// TIA Portal V15.1 export
// export: Created 2020-06-12T07:35:49.8818359Z, ExportSetting None, DisplayName Totally Integrated Automation Portal, DisplayVersion V15.1, DisplayName TIA Portal Openness, DisplayVersion V15.1, DisplayName STEP 7 Professional, DisplayVersion V15.1, DisplayName STEP 7 Safety, DisplayVersion V15.1, DisplayName WinCC Advanced, DisplayVersion V15.1
FUNCTION_BLOCK "MELT_PHASES_S"   // FB221, GRAPH
TITLE = S7GRAPH V5.0 FB
{ S7_Optimized_Access := 'TRUE' }
// Block comment
// stored: AcknowledgeErrorsRequired false, GraphVersion 2.0, LanguageInNetworks FBD, SetENOAutomatically false, WithAlarmHandling false
   // inherited from GRAPH_BASE
   VAR_INPUT
      INIT_SQ : Bool;
      eStart { ExternalAccessible := 'False'; ExternalVisible := 'False'; ExternalWritable := 'False'} : Bool;
      eCancel { ExternalAccessible := 'False'; ExternalVisible := 'False'; ExternalWritable := 'False'} : Bool;
      ePrepared { ExternalAccessible := 'False'; ExternalVisible := 'False'; ExternalWritable := 'False'} : Bool;
      ePause { ExternalAccessible := 'False'; ExternalVisible := 'False'; ExternalWritable := 'False'} : Bool;
      eStop { ExternalAccessible := 'False'; ExternalVisible := 'False'; ExternalWritable := 'False'} : Bool;
      eStarted { ExternalAccessible := 'False'; ExternalVisible := 'False'; ExternalWritable := 'False'} : Bool;
      eForceMT { ExternalAccessible := 'False'; ExternalVisible := 'False'; ExternalWritable := 'False'} : Bool;
      eStartHT { ExternalAccessible := 'False'; ExternalVisible := 'False'; ExternalWritable := 'False'} : Bool;
      eSlagMolten { ExternalAccessible := 'False'; ExternalVisible := 'False'; ExternalWritable := 'False'} : Bool;
      iCurrentRuns { ExternalAccessible := 'False'; ExternalVisible := 'False'; ExternalWritable := 'False'} : Bool;
      pStartDuration { ExternalAccessible := 'False'; ExternalVisible := 'False'; ExternalWritable := 'False'} : Int := 30;
      pHTDuration { ExternalAccessible := 'False'; ExternalVisible := 'False'; ExternalWritable := 'False'} : Int := 30;
   END_VAR
   VAR_OUTPUT
      qSTPhaseTime { ExternalAccessible := 'False'; ExternalVisible := 'False'; ExternalWritable := 'False'} : Real;   // stat phase actual time
      qHTPhaseTime { ExternalAccessible := 'False'; ExternalVisible := 'False'; ExternalWritable := 'False'} : Real;   // hottoping phase actual time
      qPhaseId { ExternalAccessible := 'False'; ExternalVisible := 'False'; ExternalWritable := 'False'} : Int;   // phase ID
   END_VAR
   VAR_IN_OUT
      ioPremelt { ExternalAccessible := 'False'; ExternalVisible := 'False'; ExternalWritable := 'False'} : Bool;
      ioMelting { ExternalAccessible := 'False'; ExternalVisible := 'False'; ExternalWritable := 'False'} : Bool;
      ioStartPhaseRun { ExternalAccessible := 'False'; ExternalVisible := 'False'; ExternalWritable := 'False'} : Bool;
      ioMainPhaseRun { ExternalAccessible := 'False'; ExternalVisible := 'False'; ExternalWritable := 'False'} : Bool;
      ioHTPhaseRun { ExternalAccessible := 'False'; ExternalVisible := 'False'; ExternalWritable := 'False'} : Bool;
      ioEnd { ExternalAccessible := 'False'; ExternalVisible := 'False'; ExternalWritable := 'False'} : Bool;
      ioStartPhaseDone { ExternalAccessible := 'False'; ExternalVisible := 'False'; ExternalWritable := 'False'} : Bool;
      ioMainPhaseDone { ExternalAccessible := 'False'; ExternalVisible := 'False'; ExternalWritable := 'False'} : Bool;
      ioHTPhaseDone { ExternalAccessible := 'False'; ExternalVisible := 'False'; ExternalWritable := 'False'} : Bool;
      ioPause { ExternalAccessible := 'False'; ExternalVisible := 'False'; ExternalWritable := 'False'} : Bool;
   END_VAR
   VAR
      sSlagMolten : Bool;
      sPhaseId { ExternalAccessible := 'False'; ExternalVisible := 'False'; ExternalWritable := 'False'} : SInt;
   END_VAR
   VAR_TEMP
      tStartPhaseDuration : Time;
      tHTPhaseDuration : Time;
      tVarR1 : Real;
      tPauseOn : Bool;
      tPauseOff : Bool;
      tSTPauseLockTime : DInt;
   END_VAR
BEGIN
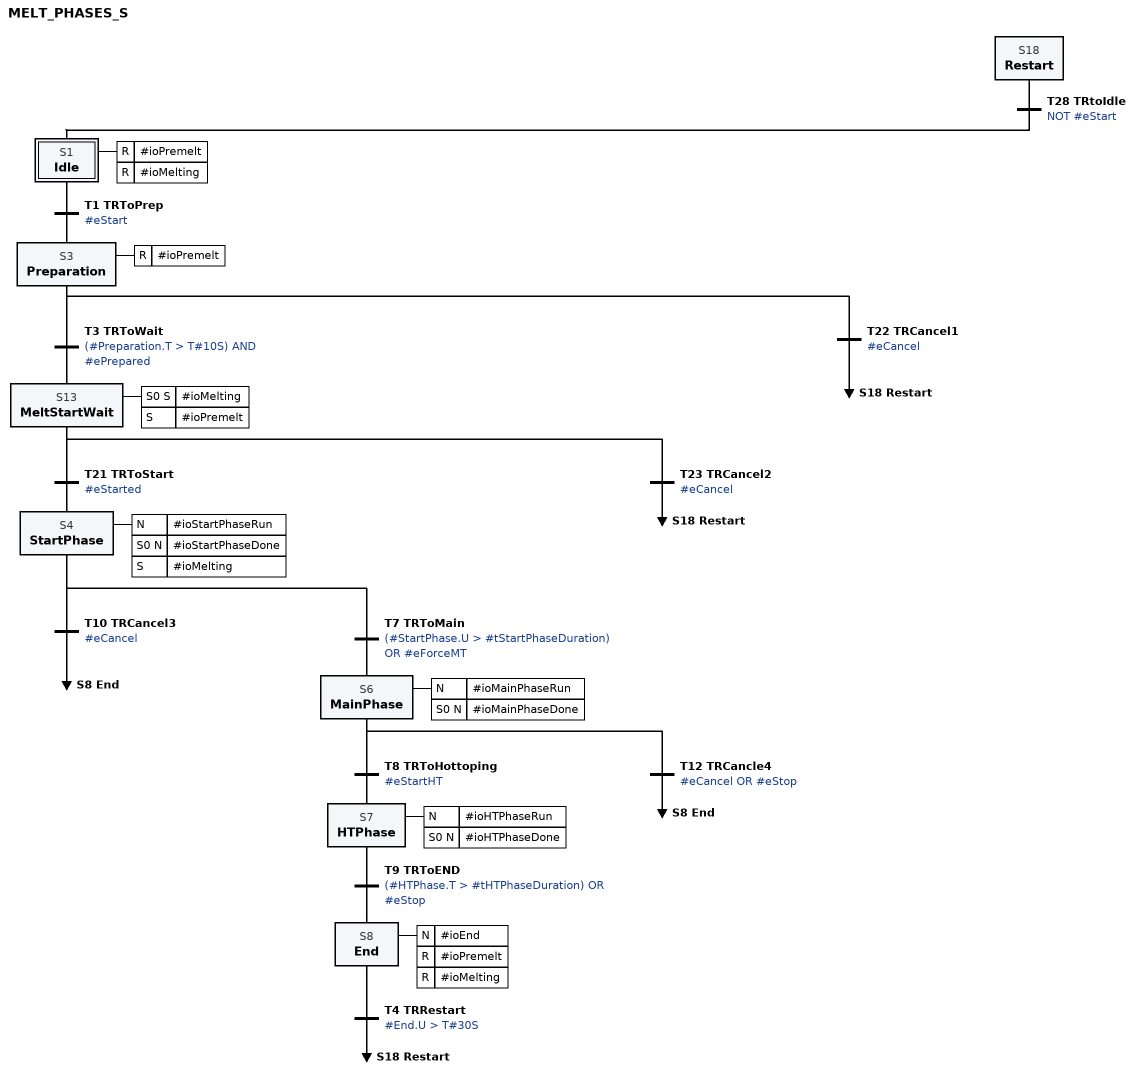
   // permanent pre-instructions
   NETWORK 1
   TITLE = Convert durations
      #tStartPhaseDuration := #pStartDuration * 60000;
      #tSTPauseLockTime := #tStartPhaseDuration / 10;
      #tHTPhaseDuration := #pHTDuration * 60000;
   NETWORK 2
   TITLE = Pause
      #tPauseOn := #ePause AND NOT #ioPause;
      #tPauseOff := (#ePause AND #ioPause) OR (NOT #StartPhase.X AND NOT #HTPhase.X) OR ((#StartPhase.T < #tSTPauseLockTime) AND #StartPhase.X);
      IF #tPauseOn THEN
          #ioPause := TRUE;   // SR flip-flop
      END_IF;
      IF #tPauseOff THEN #ioPause := FALSE; END_IF;

   // sequencer 1: Process
   INITIAL_STEP Idle:   // S1, max time T#0ms, warning time T#0ms: Step comment
      interlock C := (none);   // Idle
      supervision V := (none);   // Idle
              R    #ioPremelt
              R    #ioMelting
   END_STEP
   TRANSITION TRToPrep FROM Idle TO Preparation   // T1
      := #eStart;
   END_TRANSITION
   STEP Preparation:   // S3, max time T#0ms, warning time T#0ms: Step comment
      interlock C := (none);   // prepare
      supervision V := (none);   // prepare
              R    #ioPremelt
   END_STEP
   TRANSITION TRToWait FROM Preparation TO MeltStartWait   // T3
      := (#Preparation.T > T#10S) AND #ePrepared;
   END_TRANSITION
   TRANSITION TRCancel1 FROM Preparation TO Restart   // T22, jump
      := #eCancel;
   END_TRANSITION
   STEP StartPhase:   // S4, max time T#0ms, warning time T#0ms: Step comment
      interlock C := #iCurrentRuns AND NOT #ioPause;   // start_slag_melting
      supervision V := (none);   // start_slag_melting
              N    #ioStartPhaseRun
          S0  N    #ioStartPhaseDone
              S    #ioMelting
   END_STEP
   TRANSITION TRCancel3 FROM StartPhase TO End   // T10, jump
      := #eCancel;
   END_TRANSITION
   TRANSITION TRToMain FROM StartPhase TO MainPhase   // T7
      := (#StartPhase.U > #tStartPhaseDuration) OR #eForceMT;
   END_TRANSITION
   STEP MainPhase:   // S6, max time T#0ms, warning time T#0ms: Step comment
      interlock C := #iCurrentRuns;   // melt_phase
      supervision V := (none);   // melt_phase
              N    #ioMainPhaseRun
          S0  N    #ioMainPhaseDone
   END_STEP
   TRANSITION TRToHottoping FROM MainPhase TO HTPhase   // T8
      := #eStartHT;
   END_TRANSITION
   TRANSITION TRCancle4 FROM MainPhase TO End   // T12, jump
      := #eCancel OR #eStop;
   END_TRANSITION
   STEP HTPhase:   // S7, max time T#0ms, warning time T#0ms: Step comment
      interlock C := #iCurrentRuns AND NOT #ioPause;   // hottopping
      supervision V := (none);   // hottopping
              N    #ioHTPhaseRun
          S0  N    #ioHTPhaseDone
   END_STEP
   TRANSITION TRToEND FROM HTPhase TO End   // T9
      := (#HTPhase.T > #tHTPhaseDuration) OR #eStop;
   END_TRANSITION
   STEP End:   // S8, max time T#0ms, warning time T#0ms: Step comment
      interlock C := (none);   // end
      supervision V := (none);   // end
              N    #ioEnd
              R    #ioPremelt
              R    #ioMelting
   END_STEP
   TRANSITION TRRestart FROM End TO Restart   // T4, jump
      := #End.U > T#30S;
   END_TRANSITION
   STEP MeltStartWait:   // S13, max time T#10S, warning time T#7S
          S0  S    #ioMelting
              S    #ioPremelt
   END_STEP
   TRANSITION TRToStart FROM MeltStartWait TO StartPhase   // T21
      := #eStarted;
   END_TRANSITION
   TRANSITION TRCancel2 FROM MeltStartWait TO Restart   // T23, jump
      := #eCancel;
   END_TRANSITION
   STEP Restart:   // S18, max time T#10S, warning time T#7S
   END_STEP
   TRANSITION TRtoIdle FROM Restart TO Idle   // T28
      := NOT #eStart;
   END_TRANSITION

   // permanent post-instructions
   NETWORK 1
   TITLE = Convert actual durations
      #tVarR1 := DINT_TO_REAL(#StartPhase.U);
      IF #ioMelting THEN #qSTPhaseTime := #tVarR1 / 60000.0; END_IF;
      IF NOT #ioMelting THEN #qSTPhaseTime := 0.0; END_IF;
   NETWORK 2
   TITLE = Convert actual durations
      #tVarR1 := DINT_TO_REAL(#HTPhase.U);
      IF #HTPhase.X OR #End.X THEN #qHTPhaseTime := #tVarR1 / 60000.0; END_IF;
      IF NOT (#HTPhase.X OR #End.X) THEN #qHTPhaseTime := 0.0; END_IF;
   NETWORK 3
      IF #StartPhase.X AND #eSlagMolten THEN
          #sSlagMolten := TRUE;   // SR flip-flop
      END_IF;
      IF #Idle.X OR #End.X THEN #sSlagMolten := FALSE; END_IF;
   NETWORK 4
      #sPhaseId := 0;
      IF #Idle.X THEN #sPhaseId := 1; END_IF;
      IF #Preparation.X THEN #sPhaseId := 2; END_IF;
      IF #MeltStartWait.X THEN #sPhaseId := 3; END_IF;
      IF #StartPhase.X THEN #sPhaseId := 4; END_IF;
      IF #sSlagMolten THEN #sPhaseId := 5; END_IF;
      IF #MainPhase.X THEN #sPhaseId := 6; END_IF;
      IF #HTPhase.X THEN #sPhaseId := 7; END_IF;
      IF #End.X THEN #sPhaseId := 8; END_IF;
      #qPhaseId := #sPhaseId;
END_FUNCTION_BLOCK
